{attribute 'linkalways'} 
{attribute 'no_explicit_call' := 'This FB is a CLASS and must be accessed using methods or properties'}
{attribute 'enable_dynamic_creation'}
FUNCTION_BLOCK PUBLIC ListNode EXTENDS Disposable IMPLEMENTS I_ListNode
VAR
	pBuffer : POINTER TO BYTE;
	bufferSize : UDINT;
END_VAR

METHOD PRIVATE CopyBufferToDestination
VAR_INPUT
	DestinationAddress : PVOID;
END_VAR
MEMCPY(DestinationAddress, pBuffer, bufferSize);
END_METHOD

METHOD PRIVATE CopySourceToBuffer
VAR_INPUT
	SourceAddress : PVOID;
END_VAR
MEMCPY(pBuffer, SourceAddress, bufferSize);
END_METHOD

METHOD PRIVATE CreateBuffer
VAR_INPUT
	SizeInBytes : UDINT;
END_VAR
bufferSize := SizeInBytes;
pBuffer := __NEW(BYTE, SizeInBytes);
END_METHOD

PROPERTY PUBLIC DataSize : UDINT
GET
DataSize := bufferSize;
END_GET
END_PROPERTY

METHOD PRIVATE DestroyBuffer
VAR_INPUT
END_VAR
IF pBuffer = 0 THEN
	RETURN;
END_IF

__DELETE(pBuffer);
bufferSize := 0;
END_METHOD

METHOD PUBLIC Equals : BOOL
VAR_INPUT
	Symbol : ANY;
END_VAR
IF pBuffer = 0 THEN
	RETURN;
END_IF

IF bufferSize <> DINT_TO_UDINT(Symbol.diSize) THEN
	RETURN;
END_IF

Equals := memcmp(Symbol.pValue, pBuffer, bufferSize) = 0;
END_METHOD

METHOD FB_exit : BOOL
VAR_INPUT
	bInCopyCode : BOOL; // if TRUE, the exit method is called for exiting an instance that is copied afterwards (online change).
END_VAR
IF bInCopyCode THEN
	RETURN;
END_IF

DestroyBuffer();
END_METHOD

METHOD FB_init : BOOL
VAR_INPUT
	bInitRetains : BOOL; // if TRUE, the retain variables are initialized (warm start / cold start)
	bInCopyCode : BOOL;  // if TRUE, the instance afterwards gets moved into the copy code (online change)
	Source : ANY;
END_VAR
CreateBuffer(DINT_TO_UDINT(Source.diSize));
CopySourceToBuffer(Source.pValue);
END_METHOD

METHOD TryGet : BOOL
VAR_INPUT
	Destination	: ANY;
END_VAR
TryGet := TryGetTo(Destination.pValue, DINT_TO_UDINT(Destination.diSize));
END_METHOD

METHOD TryGetTo : BOOL
VAR_INPUT
	DestinationAddress : PVOID;
	DestinationSize : UDINT;
END_VAR
IF pBuffer = 0 THEN
	RETURN;
END_IF

IF bufferSize <> DestinationSize THEN
	RETURN;
END_IF

CopyBufferToDestination(DestinationAddress);
TryGetTo := TRUE;
END_METHOD

END_FUNCTION_BLOCK

(* stored: Version 1.1.0.1, ProductVersion 3.1.4024.12
   POU ListNode: Id {04e5c5d1-dd5d-47ab-b4f6-3475e155c010}, SpecialFunc None
   Folder Constructor: Id {826c9f1a-1cc1-46fc-b0af-b5c9123bc59f}
   Folder Destructor: Id {117fd6fe-74ef-40cb-93a2-fbf96a6821d7}
   Folder Private: Id {ad978085-9df9-4eae-8dc8-014d510715b2}
   Method CopyBufferToDestination: Id {3dba3b3a-1b4b-4b76-b407-65ece2daef65}
   Method CopySourceToBuffer: Id {08222928-3fe2-4559-af7d-3dd180f076f1}
   Method CreateBuffer: Id {ef5e76d1-6f88-4dbe-8c69-fe6d45ff059a}
   Property DataSize: Id {52a70dbb-b92e-481e-9e64-f90d005a3ac9}
   Get Get: Id {574f4209-ad6e-483b-b84c-9610c10f74d4}
   Method DestroyBuffer: Id {4ed70f4f-4840-48da-bbee-f1b2190add5c}
   Method Equals: Id {0ca78a5a-a9c9-432f-97bc-c199a16a59b5}
   Method FB_exit: Id {52762cf6-3527-4224-b13f-6b8424a2ae5d}
   Method FB_init: Id {5fc37224-f5fe-4cfc-a79a-ade4bfffe83b}
   Method TryGet: Id {49140141-1297-454f-9079-ed7a98a15421}
   Method TryGetTo: Id {f10d13c2-d6a0-43f9-8e86-471ac54f284c} *)
